// TIA Portal V16 export
// export: Created 2023-03-29T11:04:58.6238927Z, ExportSetting WithDefaults, DisplayName Totally Integrated Automation Portal, DisplayVersion V16 Update 6, DisplayName TIA Portal Version Control Interface, DisplayVersion V16 Update 2, DisplayName TIA Portal Openness, DisplayVersion V16 Update 6, DisplayName STEP 7 Professional, DisplayVersion V16 Update 6, DisplayName STEP 7 Safety, DisplayVersion V16, DisplayName WinCC Advanced, DisplayVersion V16 Update 6
DATA_BLOCK "dbControl without inverter"   // DB76
AUTHOR : rtecmer
VERSION : 0.1
// stored: AutoNumber true, DBAccessibleFromOPCUA true, InstanceOfName Sterowania bez falownika, InstanceOfType FB
"Sterowania bez falownika"
   // VAR_INPUT
   //    IsReadyP1 : Bool;
   //    IsReadyP2 : Bool;
   //    IsReadyP3 : Bool;
   //    IsReadyP4 : Bool;
   //    IsMode_Auto : Bool;
   //    InputWarning_H_PID : Bool;
   //    InputWarning_L_PID : Bool;
   //    IsReady_Inverter : Bool;
   //    PV_max : Real;
   //    Act_B3ciśnienie : Real;
   //    Rst_Driver_Max_presure : Bool;
   // END_VAR
   // VAR_OUTPUT
   //    CMD_A_Network_P1 : Bool;
   //    CMD_A_Network_P2 : Bool;
   //    CMD_A_Network_P3 : Bool;
   //    CMD_A_Network_P4 : Bool;
   // END_VAR
   // VAR
   //    stc_PV : Real;
   // END_VAR
BEGIN
END_DATA_BLOCK
